# EPICS StreamDevice protocol: docker/PSAppTest/PS_DB/tc-l2s.proto
OutTerminator = CR LF;
InTerminator  = LF;

readDOR {
  out "@DOR?";
  in "%5c";
}

readDIR {
  out "@DIR?";
  in "%5c";
}

setDOR {
  out "@DO%02u";
  in "%5c"
}

setADDR {
  out "ADDRess %u";
  in "%s"
}
